FUNCTION_BLOCK load (* ODE *)
  (* Standard: 61499-2 *)
  (* Version 0.1, 2017-00-25, hpea485, UOA *)
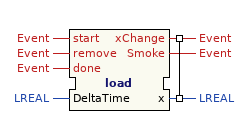
  EVENT_INPUT
    start;
    remove;
    done;
  END_EVENT
  EVENT_OUTPUT
    xChange WITH x;
    Smoke;
  END_EVENT
  VAR_INPUT
    DeltaTime : LREAL := 0.01;
  END_VAR
  VAR_OUTPUT
    x : LREAL;
  END_VAR
  VAR
    i_fault : LREAL := 800.0;
    i_inrush : LREAL := 800.0;
    t_up : LREAL := 0.2;
    t_down : LREAL := 0.4;
    i_nom : LREAL := 200.0;
  END_VAR
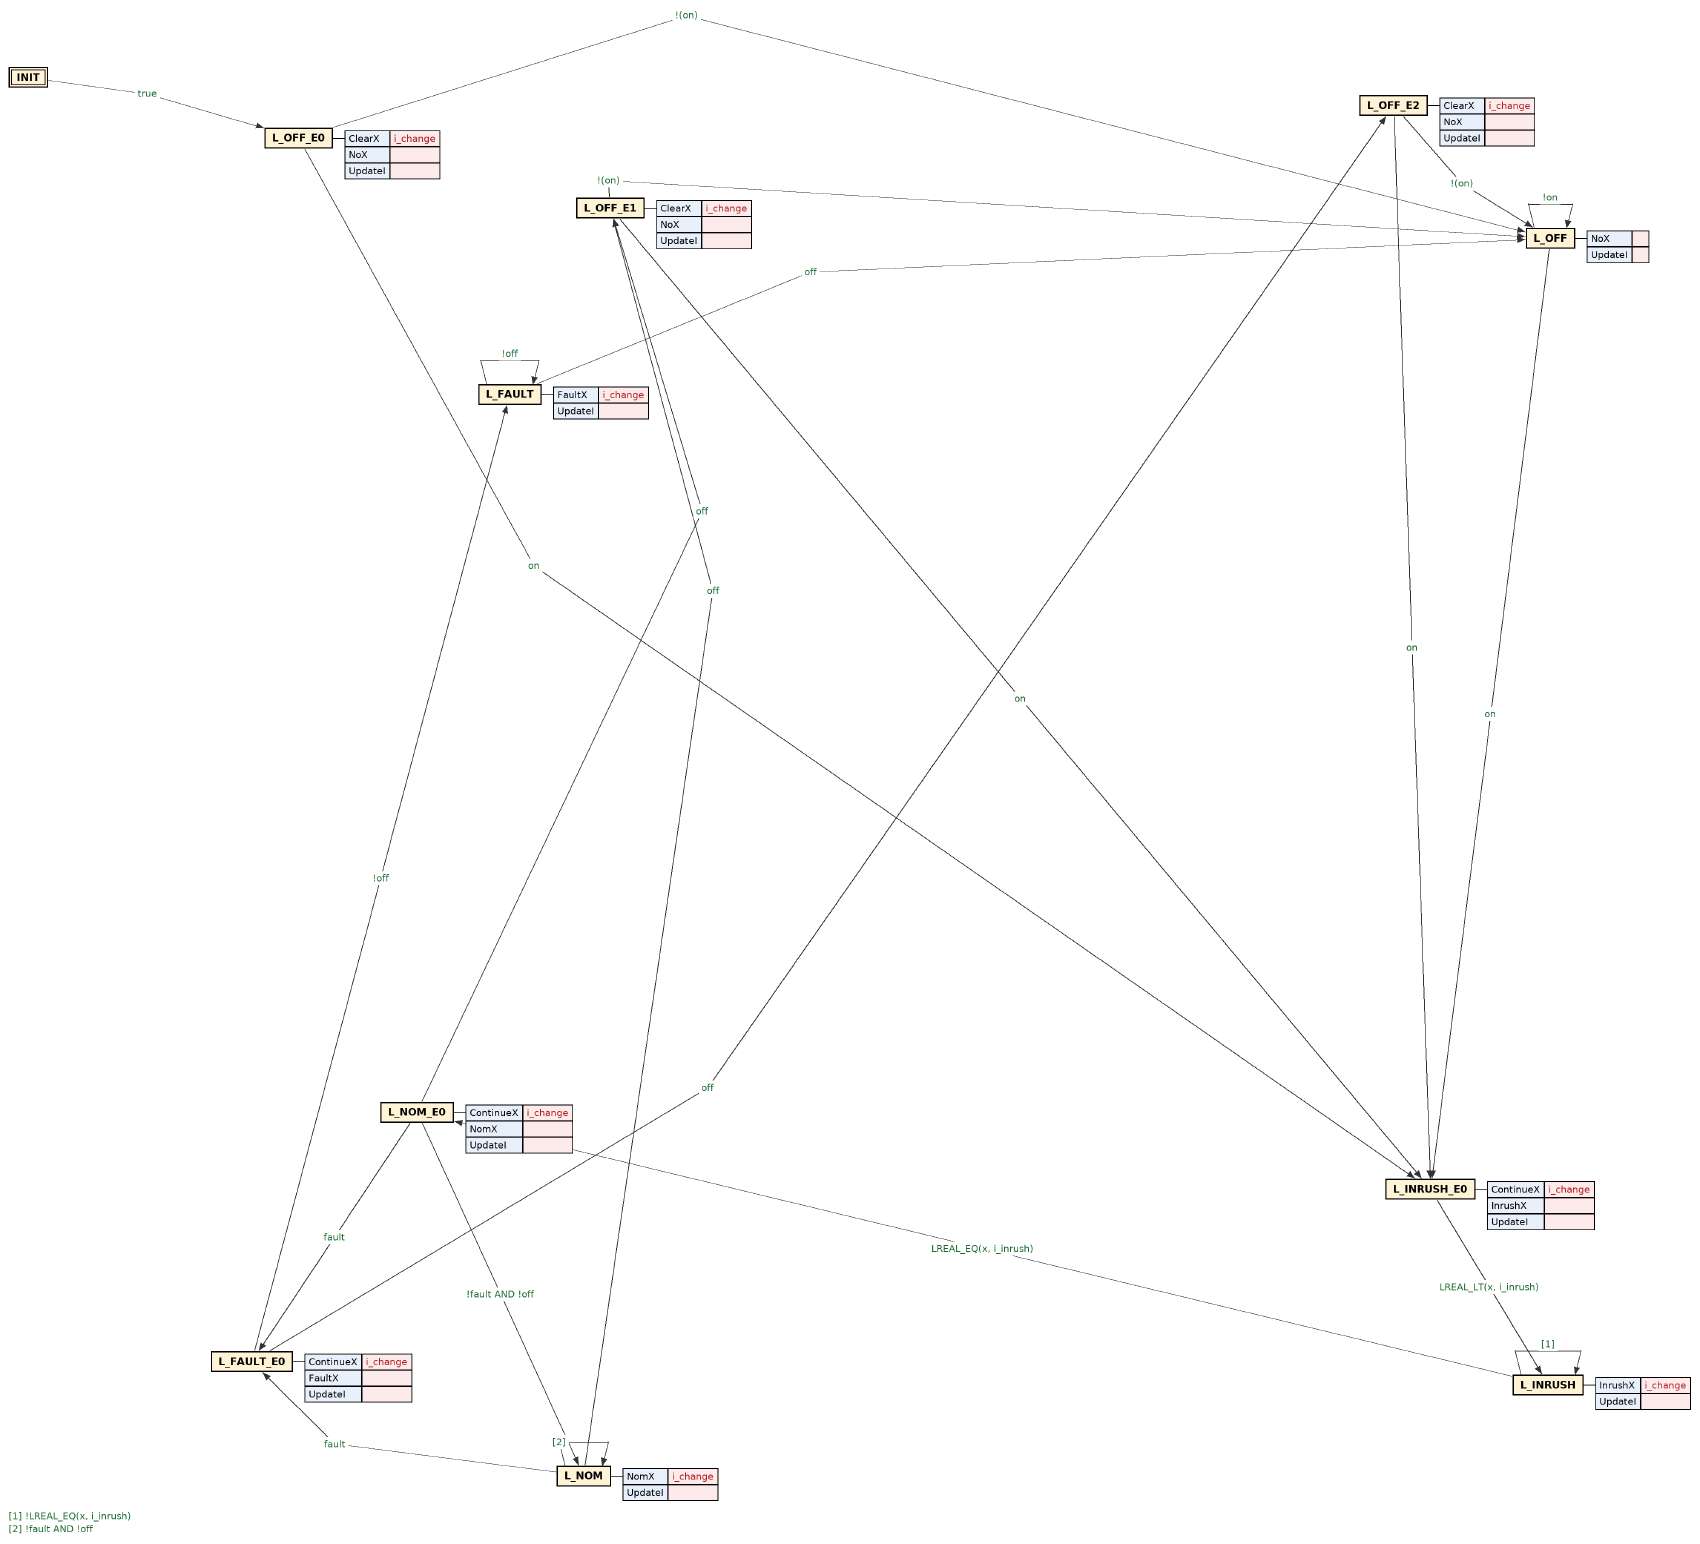
  EC_STATES
    INIT;
    L_OFF_E0 : ClearX -> i_change, NoX, UpdateI;
    L_OFF_E1 : ClearX -> i_change, NoX, UpdateI;
    L_OFF_E2 : ClearX -> i_change, NoX, UpdateI;
    L_OFF : NoX, UpdateI;
    L_INRUSH_E0 : ContinueX -> i_change, InrushX, UpdateI;
    L_INRUSH : InrushX -> i_change, UpdateI;
    L_NOM_E0 : ContinueX -> i_change, NomX, UpdateI;
    L_NOM : NomX -> i_change, UpdateI;
    L_FAULT_E0 : ContinueX -> i_change, FaultX, UpdateI;
    L_FAULT : FaultX -> i_change, UpdateI;
  END_STATES
  EC_TRANSITIONS
    INIT TO L_OFF_E0 := true;
    L_OFF_E0 TO L_OFF := !(on);
    L_OFF_E0 TO L_INRUSH_E0 := on;
    L_OFF_E1 TO L_OFF := !(on);
    L_OFF_E1 TO L_INRUSH_E0 := on;
    L_OFF_E2 TO L_OFF := !(on);
    L_OFF_E2 TO L_INRUSH_E0 := on;
    L_OFF TO L_INRUSH_E0 := on;
    L_OFF TO L_OFF := !on;
    L_INRUSH_E0 TO L_NOM_0 := LREAL_EQ(x, i_inrush);
    L_INRUSH_E0 TO L_INRUSH := LREAL_LT(x, i_inrush);
    L_INRUSH TO L_NOM_E0 := LREAL_EQ(x, i_inrush);
    L_INRUSH TO L_INRUSH := !LREAL_EQ(x, i_inrush);
    L_NOM_E0 TO L_NOM := !fault AND !off;
    L_NOM_E0 TO L_OFF_E1 := off;
    L_NOM_E0 TO L_FAULT_E0 := fault;
    L_NOM TO L_OFF_E1 := off;
    L_NOM TO L_FAULT_E0 := fault;
    L_NOM TO L_NOM := !fault AND !off;
    L_FAULT_E0 TO L_OFF_E2 := off;
    L_FAULT_E0 TO L_FAULT := !off;
    L_FAULT TO L_OFF := off;
    L_FAULT TO L_FAULT := !off;
  END_TRANSITIONS
  ALGORITHM ClearX IN C: (* ODE_init *)
x_prime = 0;
  END_ALGORITHM
  ALGORITHM ContinueX IN C: (* ODE_init *)
x_prime = x;
  END_ALGORITHM
  ALGORITHM NoX IN C: (* ODE *)
x_dot = 0;
  END_ALGORITHM
  ALGORITHM InrushX IN C: (* ODE *)
x_dot = (5/t_up)*(i_inrush*1.01 - x);
x_trigger = i_inrush;
  END_ALGORITHM
  ALGORITHM NomX IN C: (* ODE *)
x_dot = (5/t_down)*(i_nom - x);
  END_ALGORITHM
  ALGORITHM FaultX IN C: (* ODE *)
x_dot =  (5/t_fault) * (i_fault - x);
  END_ALGORITHM
  ALGORITHM UpdateI IN C:
me->i = me->x;
  END_ALGORITHM
END_FUNCTION_BLOCK
